PROGRAM MAIN
VAR
END_VAR

END_PROGRAM

(* stored: Version 1.1.0.1
   POU MAIN: Id {eefb6ac3-74a0-4af3-86ef-b9841645e639} *)
